Yaskawa INFORM job: SYS_SPINDLE_STOP.JBI

/JOB
//NAME SYS_SPINDLE_STOP
//POS
///NPOS 0,0,0,0,0,0
//INST
///DATE 2021/12/03 11:59
///ATTR SC,RW
///GROUP1 RB1
NOP
DOUT OT#(1) OFF
WAIT T=7.00
DOUT OT#(17) OFF
END
